// TwinCAT 3 PLC project TcoPneumatics
// Title: TcoPneumatics
// Company: Vortex.Library
// Author: Dustin Hullett
// ProjectVersion: 0.1.0.88
// ProgramVersion: 3.1.4023.0
// libraries:
//   Tc2_Standard, * (Beckhoff Automation GmbH)
//   Tc2_System, * (Beckhoff Automation GmbH)
//   Tc3_Module, * (Beckhoff Automation GmbH)
// project tree:
//   ComponentsBase/ fbComponent.TcPOU
//   GVLs/ IO.TcGVL (not stored)
//   / PlcTask.TcTTO
//   POUs/Cylinders/ fbCylinder.TcPOU, ICylinder.TcIO
//   POUs/HW/Beckhoff/EL922x/FBs/ FuseChannelBasic.TcPOU, FuseChannelExtended.TcPOU, FuseModuleEL922x.TcPOU
//   POUs/HW/Beckhoff/EL922x/ITFs/ IFuseChannelBasic.TcIO, IFuseChannelExtended.TcIO
//   POUs/HW/Beckhoff/EL922x/STs/ EL922x_ChannelBasic.TcDUT, EL922x_ChannelExtended.TcDUT, OutputStruct.TcDUT, StatusStructBasic.TcDUT, StatusStructExtended.TcDUT
//   POUs/ MAIN.TcPOU
//   Tasks/ eTaskState.TcDUT (not stored), fbTask.TcPOU (not stored), ITaskContainer.TcIO (not stored), ITaskStatus.TcIO
//   Version/ Global_Version.TcGVL (not stored)
//   _Tests/ MAIN_TESTS.TcPOU
//   _Tests/Tasks/ fbTaskTests.TcPOU (not stored)
// real-time tasks:
//   TASK PlcTask: cycle T#10ms, priority 20, ADS port 350

CONFIGURATION TcoPneumatics
    RESOURCE PLC ON TwinCAT3
        TASK PlcTask(INTERVAL := T#10ms, PRIORITY := 20);
        PROGRAM MAIN WITH PlcTask : MAIN;
    END_RESOURCE
END_CONFIGURATION

// ---- POUs/HW/Beckhoff/EL922x/STs/EL922x_ChannelBasic.TcDUT
TYPE EL922x_ChannelBasic :
STRUCT
	Status AT%I* : StatusStructBasic;
	Control AT%q* : OutputStruct;
END_STRUCT
END_TYPE

// ---- POUs/HW/Beckhoff/EL922x/STs/EL922x_ChannelExtended.TcDUT
TYPE EL922x_ChannelExtended :
STRUCT
	Status AT%I* : StatusStructExtended;
	Load AT%I* : UINT;
	Current AT%I* : UINT;
	VoltageIn AT%I* : UINT;
	VoltageOut AT%I* : UINT;
	Control AT%q* : OutputStruct;
END_STRUCT
END_TYPE

// ---- POUs/HW/Beckhoff/EL922x/STs/OutputStruct.TcDUT
TYPE OutputStruct :
STRUCT
	Reset : BIT;
	Switch	 : BIT;
	{attribute 'hide'}
	_hidden_bit_0: BIT;
	{attribute 'hide'}
	_hidden_bit_1: BIT;
	{attribute 'hide'}
	_hidden_bit_2: BIT;
	{attribute 'hide'}
	_hidden_bit_3: BIT;
	{attribute 'hide'}
	_hidden_bit_4: BIT;
	{attribute 'hide'}
	_hidden_bit_5: BIT;
	{attribute 'hide'}
	_hidden_byte_0: BYTE;
END_STRUCT
END_TYPE

// ---- POUs/HW/Beckhoff/EL922x/STs/StatusStructBasic.TcDUT
TYPE StatusStructBasic :
STRUCT
		Enabled: BIT;
		Tripped : BIT;
		{attribute 'hide'}
		_hidden_bit_0: BIT;
		{attribute 'hide'}
		_hidden_bit_1: BIT;
		HWProtection : BIT;
		{attribute 'hide'}
		_hidden_bit_2: BIT;
		{attribute 'hide'}
		_hidden_bit_3: BIT;
		CurrentLevelWarning : BIT;
		
		CoolDownLock : BIT;
		{attribute 'hide'}
		_hidden_bit_4: BIT;
		{attribute 'hide'}
		_hidden_bit_5: BIT;
		{attribute 'hide'}
		_hidden_bit_6: BIT;
		Diag : BIT;
		TxPDOState : BIT;
		{attribute 'hide'}
		_hidden_bit_7: BIT;
		{attribute 'hide'}
		_hidden_bit_8: BIT;
		
		{attribute 'hide'}
		_hidden_bit_9: BIT;
		{attribute 'hide'}
		_hidden_bit_10: BIT;
		Error : BIT;
		StateReset : BIT;
		StateSwitch : BIT;
		{attribute 'hide'}
		_hidden_bit_11: BIT;
		{attribute 'hide'}
		_hidden_bit_12: BIT;
		{attribute 'hide'}
		_hidden_bit_13: BIT;
		{attribute 'hide'}
		_hidden_byte_14: BYTE;
END_STRUCT
END_TYPE

// ---- POUs/HW/Beckhoff/EL922x/STs/StatusStructExtended.TcDUT
TYPE StatusStructExtended :
STRUCT
	Enabled: BIT;
	Tripped : BIT;
	ShortCircuit : BIT;
	Overload : BIT;
	HWProtection : BIT;
	Overvoltage : BIT;
	Undervoltage : BIT;
	CurrentLevelWarning : BIT;
	
	CoolDownLock : BIT;
	DisabledBySwitch : BIT;
	DisabledByDI : BIT;
	DisabledByOutput : BIT;
	Diag : BIT;
	TxPDOState : BIT;
	InputCycleCount : BIT;
	InputCycleCount2 : BIT;
	
	StateDeviceSwitch : BIT;
	StateDigitalInput : BIT;
	Error : BIT;
	StateReset : BIT;
	StateSwitch : BIT;
	{attribute 'hide'}
	_hidden_bit_0: BIT;
	{attribute 'hide'}
	_hidden_bit_1: BIT;
	{attribute 'hide'}
	_hidden_bit_2: BIT;
	{attribute 'hide'}
	_hidden_byte_0: BYTE;
END_STRUCT
END_TYPE

// ---- POUs/Cylinders/ICylinder.TcIO
INTERFACE ICylinder EXTENDS __System.IQueryInterface

PROPERTY AtHome : bool
GET
END_GET
END_PROPERTY

PROPERTY AtWork : bool
GET
END_GET
END_PROPERTY

METHOD MoveToHome : ITaskStatus
END_METHOD

METHOD MoveToWork : ITaskStatus
END_METHOD

END_INTERFACE

// ---- POUs/HW/Beckhoff/EL922x/ITFs/IFuseChannelBasic.TcIO
INTERFACE IFuseChannelBasic EXTENDS __SYSTEM.IQueryInterface

PROPERTY CoolDownLock  : bool
GET
END_GET
END_PROPERTY

PROPERTY CurrentLevelWarning  : bool
GET
END_GET
END_PROPERTY

PROPERTY Diag  : bool
GET
END_GET
END_PROPERTY

PROPERTY Enabled : bool
GET
END_GET
END_PROPERTY

PROPERTY Error  : bool
GET
END_GET
END_PROPERTY

PROPERTY HardwareProtection : bool
GET
END_GET
END_PROPERTY

METHOD ResetFuse : BOOL
END_METHOD

PROPERTY StateReset : bool
GET
END_GET
END_PROPERTY

PROPERTY StateSwitch : bool
GET
END_GET
END_PROPERTY

METHOD SwitchFuse : BOOL
END_METHOD

PROPERTY Tripped : bool
GET
END_GET
END_PROPERTY

PROPERTY TxPDOState  : bool
GET
END_GET
END_PROPERTY

END_INTERFACE

// ---- POUs/HW/Beckhoff/EL922x/ITFs/IFuseChannelExtended.TcIO
INTERFACE IFuseChannelExtended EXTENDS __SYSTEM.IQueryInterface

PROPERTY DisabledByDI : BOOL
GET
END_GET
END_PROPERTY

PROPERTY DisabledByOutput : BOOL
GET
END_GET
END_PROPERTY

PROPERTY DisabledBySwitch : BOOL
GET
END_GET
END_PROPERTY

PROPERTY Overload : BOOL
GET
END_GET
END_PROPERTY

PROPERTY Overvoltage : BOOL
GET
END_GET
END_PROPERTY

PROPERTY ShortCircuit : BOOL
GET
END_GET
END_PROPERTY

PROPERTY StateDeviceSwitch : BOOL
GET
END_GET
END_PROPERTY

PROPERTY StateDigitalInput : BOOL
GET
END_GET
END_PROPERTY

PROPERTY Undervoltage : BOOL
GET
END_GET
END_PROPERTY

END_INTERFACE

// ---- Tasks/ITaskStatus.TcIO
INTERFACE ITaskStatus

METHOD Abort
END_METHOD

PROPERTY Busy : BOOL
GET
END_GET
END_PROPERTY

PROPERTY Done : BOOL
GET
END_GET
END_PROPERTY

PROPERTY Error : BOOL
GET
END_GET
END_PROPERTY

END_INTERFACE

// ---- POUs/MAIN.TcPOU
PROGRAM MAIN
VAR	
	{attribute wpf [Container(Layout.Stack)]}	
	{attribute addProperty Name "WPF cyclinder"}
	_wpfCyclinder : fbCylinder;	
	{attribute wpf [Container(Layout.Stack)]}	
	{attribute addProperty Name "WPF cyclinder 1"}
	_wpfCyclinder_1 : fbCylinder;
	{attribute wpf [Container(Layout.Stack)]}	
	{attribute addProperty Name "WPF cyclinder 2"}
	_wpfCyclinder_2 : fbCylinder;
	{attribute wpf [Container(Layout.Stack)]}	
	{attribute addProperty Name "WPF cyclinder 3"}
	_wpfCyclinder_3 : fbCylinder;	
END_VAR

_wpfCyclinder(inAtHomePos:=IO.A1[0] , inAtWorkPos:=IO.A1[1] , outToHomePos=> IO.A2[0], outToWorkPos=>IO.A2[1]);

MAIN_TESTS();

END_PROGRAM

// ---- POUs/Cylinders/fbCylinder.TcPOU
FUNCTION_BLOCK fbCylinder EXTENDS fbComponent IMPLEMENTS ICylinder
VAR_INPUT
	(*~
		<docu>
			<summary>
				Home position sensor.
			</summary>	
		</docu>
	~*)
	{attribute wpf [Container(Layout.UniformGrid)]}
	{attribute wpf [Group(Layout.GroupBox, "Inputs")]}	
	{attribute addProperty Name "Home position sensor"}
	inAtHomePos : BOOL;
	(*~
		<docu>
			<summary>
				Working position sensor.
			</summary>	
		</docu>
	~*) 
	{attribute addProperty Name "Work position sensor"}
	inAtWorkPos : BOOL; 
END_VAR
VAR_OUTPUT
	(*~
		<docu>
			<summary>
				Move to working home position signal.
			</summary>	
		</docu>
	~*)
	{attribute wpf [Container(Layout.UniformGrid)]}
	{attribute wpf [Group(Layout.GroupBox, "Outputs")]}	
	{attribute addProperty Name "Move to home position actuator"}
	outToHomePos : BOOL;
	(*~
		<docu>
			<summary>
				Move to working posistion signal.
			</summary>	
		</docu>
	~*)
	{attribute addProperty Name "Move to work position actuator"}
	outToWorkPos : BOOL;
	
	haha : BOOL;
END_VAR

VAR	
	{attribute wpf [Container(Layout.UniformGrid)]}
	{attribute addProperty Name "Request move to Home position"}	
	_moveHomeTask : fbTask(THIS^);
	{attribute addProperty Name "Request move to Work position"}
	_moveWorkTask : fbTask(THIS^);
	{attribute addProperty Name "Request Stop"}
	_stopTask : fbTask(THIS^);
END_VAR

IF(_moveHomeTask.Execute(1)) THEN
	outToHomePos := TRUE;
	outToWorkPos := FALSE; 		
	_moveHomeTask.DoneWhen(inAtHomePos);			
END_IF

IF(_moveWorkTask.Execute(2)) THEN
	outToWorkPos := TRUE; 
	outToHomePos := FALSE;
	_moveWorkTask.DoneWhen(inAtWorkPos);
END_IF;	 

IF(_stopTask.Execute(0)) THEN	
	outToWorkPos := FALSE; 
	outToHomePos := FALSE;
	_moveWorkTask.Reset();
	_moveHomeTask.Reset();
	_stopTask.Reset();
	_stopTask.DoneWhen(TRUE);	
END_IF

{attribute 'TcRpcEnable'}
METHOD INTERNAL _MoveToHomeTest : BOOL
_MoveToHomeTest := MoveToHome().Done;
END_METHOD

{attribute 'TcRpcEnable'}
METHOD INTERNAL _MoveToWorkTest : BOOL
_MoveToWorkTest := MoveToWork().Done;
END_METHOD

{attribute 'TcRpcEnable'}
METHOD INTERNAL _StopTest : BOOL
_StopTest := Stop().Done;
END_METHOD

PROPERTY AtHome : bool
GET
AtHome := inAtHomePos;
END_GET
END_PROPERTY

PROPERTY AtWork : bool
GET
AtWork := inAtWorkPos;
END_GET
END_PROPERTY

METHOD PROTECTED  ManualControl
END_METHOD

(*~
	<docu>
		<summary>
			Moves the piston into home position.
		</summary>
		<returns>True when home position sensor is reached.</returns>
	</docu>
~*)
METHOD MoveToHome : ITaskStatus
THIS^._moveHomeTask.Invoke();
MoveToHome := THIS^._moveHomeTask;
END_METHOD

(*~
	<docu>
		<summary>
			Moves the piston into working position.
		</summary>
		<returns>True when working position sensor is reached.</returns>
	</docu>
~*)
METHOD MoveToWork : ITaskStatus
THIS^._moveWorkTask.Invoke();
MoveToWork := THIS^._moveWorkTask;
END_METHOD

METHOD Stop : REFERENCE TO fbTask
_stopTask.Invoke();
Stop REF= _stopTask;
END_METHOD

END_FUNCTION_BLOCK

// ---- ComponentsBase/fbComponent.TcPOU
FUNCTION_BLOCK ABSTRACT fbComponent IMPLEMENTS ITaskContainer
VAR	
	{attribute addProperty Name "Components' message"}
	{attribute clr [ReadOnly()]}
	_message : STRING(255);
	{attribute 'hide'}
	_lock : INT;		
END_VAR

METHOD PROTECTED Info
VAR_INPUT
	inMessage : STRING(255);
END_VAR
_message := inMessage;
END_METHOD

PROPERTY Lock : INT
GET
Lock := _lock;
END_GET
SET
_lock := Lock;
END_SET
END_PROPERTY

METHOD PUBLIC Manual
THIS^.ManualControl();
END_METHOD

METHOD PROTECTED ABSTRACT ManualControl
END_METHOD

END_FUNCTION_BLOCK

// ---- _Tests/MAIN_TESTS.TcPOU
PROGRAM INTERNAL MAIN_TESTS
VAR
	_taskTests : fbTaskTests;
END_VAR

_taskTests();

END_PROGRAM

// ---- POUs/HW/Beckhoff/EL922x/FBs/FuseChannelBasic.TcPOU
FUNCTION_BLOCK FuseChannelBasic IMPLEMENTS IFuseChannelBasic
VAR_INPUT
END_VAR
VAR_OUTPUT
END_VAR
VAR
	_Chn : EL922x_ChannelBasic;
END_VAR


PROPERTY CoolDownLock : BOOL
GET
CoolDownLock := _Chn.Status.CoolDownLock;
END_GET
END_PROPERTY


PROPERTY CurrentLevelWarning : BOOL
GET
CurrentLevelWarning := _Chn.Status.CurrentLevelWarning;
END_GET
END_PROPERTY


PROPERTY Diag : BOOL
GET
Diag := _Chn.Status.Diag;
END_GET
END_PROPERTY


PROPERTY Enabled : BOOL
GET
Enabled := _Chn.Status.Enabled;
END_GET
END_PROPERTY


PROPERTY Error : BOOL
GET
Error := _Chn.Status.Error;
END_GET
END_PROPERTY


PROPERTY HardwareProtection : BOOL
GET
HardwareProtection := _Chn.Status.HWProtection;
END_GET
END_PROPERTY


METHOD ResetFuse : BOOL
_Chn.Control.Reset := NOT _Chn.Control.Reset;
END_METHOD


PROPERTY StateReset : BOOL
GET
StateReset := _Chn.Status.StateReset;
END_GET
END_PROPERTY


PROPERTY StateSwitch : BOOL
GET
StateSwitch := _Chn.Status.StateSwitch;
END_GET
END_PROPERTY

METHOD SwitchFuse : BOOL
_Chn.Control.Switch := NOT _Chn.Control.Switch;
END_METHOD


PROPERTY Tripped : BOOL
GET
Tripped := _Chn.Status.Tripped;
END_GET
END_PROPERTY


PROPERTY TxPDOState : BOOL
GET
TxPDOState := _Chn.Status.TxPDOState;
END_GET
END_PROPERTY

END_FUNCTION_BLOCK

// ---- POUs/HW/Beckhoff/EL922x/FBs/FuseChannelExtended.TcPOU
FUNCTION_BLOCK FuseChannelExtended EXTENDS FuseChannelBasic IMPLEMENTS IFuseChannelExtended
VAR_INPUT
END_VAR
VAR_OUTPUT
END_VAR
VAR
	_ChnEx : EL922x_ChannelExtended;
END_VAR


PROPERTY DisabledByDI : BOOL
GET
DisabledByDI := _ChnEx.Status.DisabledByDI;
END_GET
END_PROPERTY


PROPERTY DisabledByOutput : BOOL
GET
DisabledByOutput := _ChnEx.Status.DisabledByOutput;
END_GET
END_PROPERTY


PROPERTY DisabledBySwitch : BOOL
GET
DisabledBySwitch := _ChnEx.Status.DisabledBySwitch;
END_GET
END_PROPERTY


PROPERTY Overload : BOOL
GET
Overload := _ChnEx.Status.Overload;
END_GET
END_PROPERTY


PROPERTY Overvoltage : BOOL
GET
Overvoltage := _ChnEx.Status.Overvoltage;
END_GET
END_PROPERTY

{warning 'add property implementation'}
PROPERTY ShortCircuit : BOOL
GET
ShortCircuit := _ChnEx.Status.ShortCircuit;
END_GET
END_PROPERTY

{warning 'add property implementation'}
PROPERTY StateDeviceSwitch : BOOL
GET
StateDeviceSwitch := _ChnEx.Status.StateDeviceSwitch;
END_GET
END_PROPERTY

{warning 'add property implementation'}
PROPERTY StateDigitalInput : BOOL
GET
StateDigitalInput := _ChnEx.Status.StateDigitalInput;
END_GET
END_PROPERTY

{warning 'add property implementation'}
PROPERTY Undervoltage : BOOL
GET
Undervoltage := _ChnEx.Status.Undervoltage;
END_GET
END_PROPERTY

END_FUNCTION_BLOCK

// ---- POUs/HW/Beckhoff/EL922x/FBs/FuseModuleEL922x.TcPOU
FUNCTION_BLOCK FuseModuleEL922x
VAR_INPUT
END_VAR
VAR_OUTPUT
END_VAR
VAR
	_chn1Basic : IFuseChannelBasic;
	_chn2Basic : IFuseChannelBasic;
	_chn1Extended : IFuseChannelExtended;
	_chn2Extended : IFuseChannelExtended;
END_VAR

METHOD FB_init : BOOL
VAR_INPUT
	bInitRetains : BOOL; // if TRUE, the retain variables are initialized (warm start / cold start)
	bInCopyCode : BOOL;  // if TRUE, the instance afterwards gets moved into the copy code (online change)
	chn1 : IFuseChannelBasic;
	chn2 : IFuseChannelBasic;
END_VAR
_chn1Basic := chn1;
__QUERYINTERFACE(_chn1Basic, _chn1Extended);
_chn2Basic := chn2;
__QUERYINTERFACE(_chn2Basic, _chn2Extended);
END_METHOD

END_FUNCTION_BLOCK
